// TIA Portal V20 export
VAR_GLOBAL   // PLC tag table "Default tag table"
   M_ID AT %MW10 : Int;
   EMG_Robot AT %I220.0 : Bool;
   EMG_MC1 AT %I220.1 : Bool;
   EMG_MC2 AT %I220.2 : Bool;
   EMG_OP AT %I220.3 : Bool;
   Start_AUX AT %I230.2 : Bool;
   Door_Robot_locked AT %I230.0 : Bool;
   Door_OP_locked AT %I230.1 : Bool;
   EMG_FROM_MC AT %I230.3 : Bool;
   Q_STO_Units_CH1 AT %Q260.0 : Bool;
   Q_STO_Robot_CH2 AT %Q260.3 : Bool;
   Q_Unlock_Robot_Door_1 AT %Q270.0 : Bool;
   "Q270.2" AT %Q270.2 : Bool;
   Clock_Byte AT %MB0 : Byte;
   Clock_10Hz AT %M0.0 : Bool;
   Clock_5Hz AT %M0.1 : Bool;
   "Clock_2.5Hz" AT %M0.2 : Bool;
   Clock_2Hz AT %M0.3 : Bool;
   "Clock_1.25Hz" AT %M0.4 : Bool;
   Clock_1Hz AT %M0.5 : Bool;
   "Clock_0.625Hz" AT %M0.6 : Bool;
   "Clock_0.5Hz" AT %M0.7 : Bool;
   Q_STO_Units_CH2 AT %Q260.1 : Bool;
   Q_STO_Robot_CH1 AT %Q260.2 : Bool;
   contatore AT %MW2 : Int;
   MAC1_door_open_CH1 AT %I237.0 : Bool;
   MAC1_door_open_CH2 AT %I237.1 : Bool;
   DOOR_FOR_MC_1 AT %Q275.0 : Bool;
   DOOR_FOR_MC_2 AT %Q275.1 : Bool;
   EME_PULS_MAN AT %I237.2 : Bool;
   DOOR_CLOSED AT %I237.3 : Bool;
   Q_Unlock_Robot_Door_2 AT %Q270.1 : Bool;
   Tag_4 AT %IB43 : Byte;
   Tag_5 AT %QB45 : Byte;
END_VAR
VAR_GLOBAL CONSTANT   // user constants
   _master : Int := 0;
   _Gripper_Hook_Search : Int := 16;
   _Gripper4Pallet_Search : Int := 17;
   updatePartOnTray : Int := 18;
   _Pallet_TRAY_to_Robot : Int := 1;
   _Pallet_Robot_to_TRAY : Int := 2;
   _Pallet_Robot_to_MC : Int := 3;
   _Pallet_MC_to_Robot : Int := 4;
   _Part_TRAY_to_Robot : Int := 5;
   _Part_Robot_to_TRAY : Int := 6;
   _Part_Robot_to_MC : Int := 7;
   _Part_MC_to_Robot : Int := 8;
   _Set_Gripper_OnBoard : Int := 10;
   _Vice_Robot_to_TRAY : Int := 11;
   _Vice_Robot_to_MC : Int := 12;
   _Vice_MC_to_Robot : Int := 13;
   _Gripper_TRAY_to_Robot : Int := 14;
   _Gripper_Robot_to_TRAY : Int := 15;
   Extract_TRAY : Int := 19;
   Release_TRAY : Int := 20;
   change_TCP_Data : Int := 21;
   get_TCP_Data : Int := 22;
   updateGripperOnRobot : Int := 23;
   updatePartOnRobot : Int := 24;
   updatePartOnMC : Int := 25;
   Extract_TRAY_HMI : Int := 27;
   Release_TRAY_HMI : Int := 28;
   updatePalletOnTRAY : Int := 26;
   Reset_or_log_MissionData : Int := 30;
   executeOneQuery : Int := 29;
   _Declare_Position : Int := 9;
END_VAR
